FUNCTION_BLOCK FieldsPreferredProvider (* Translate individual fields to a PreferredProvider type *)
  (* Standard: 61499-2; Description: Copyright (c) 2018 fortiss GmbH This program and the accompanying materials are made available under the terms of the Eclipse Public License 2.0 which is available at https://www.eclipse.org/legal/epl-2.0/ SPDX-License-Identifier: EPL-2.0 *)
  (* Version 1.0, 2018-09-21, Jose Cabral, fortiss GmbH *)
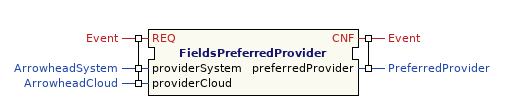
  EVENT_INPUT
    REQ WITH providerSystem, providerCloud; (* Create Preferred Provider *)
  END_EVENT
  EVENT_OUTPUT
    CNF WITH preferredProvider; (* Preferred Provider created *)
  END_EVENT
  VAR_INPUT
    providerSystem : ArrowheadSystem; (* System of the Preferred Provider *)
    providerCloud : ArrowheadCloud; (* Cloud of the Preferred Provider *)
  END_VAR
  VAR_OUTPUT
    preferredProvider : PreferredProvider; (* Preferred Provider created *)
  END_VAR
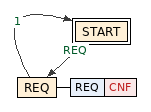
  EC_STATES
    START; (* Initial State *)
    REQ : REQ -> CNF; (* Normal execution *)
  END_STATES
  EC_TRANSITIONS
    START TO REQ := REQ;
    REQ TO START := 1;
  END_TRANSITIONS
  ALGORITHM REQ IN ST: (* Normally executed algorithm *)
preferredProvider.providerSystem := providerSystem;
preferredProvider.providerCloud := providerCloud;
  END_ALGORITHM
END_FUNCTION_BLOCK
